RESOURCE_TYPE topCFB1
  (* Standard: 61499-2 *)
  (* Version 0.1, 2017-00-09, Hammond, HAMMONDSDESKTOP *)
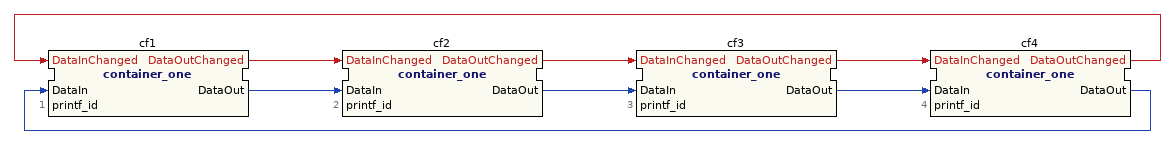
  FBS
    cf1 : container_one(printf_id := 1);
    cf2 : container_one(printf_id := 2);
    cf3 : container_one(printf_id := 3);
    cf4 : container_one(printf_id := 4);
  END_FBS
  EVENT_CONNECTIONS
    cf1.DataOutChanged TO cf2.DataInChanged;
    cf2.DataOutChanged TO cf3.DataInChanged;
    cf3.DataOutChanged TO cf4.DataInChanged;
    cf4.DataOutChanged TO cf1.DataInChanged;
  END_CONNECTIONS
  DATA_CONNECTIONS
    cf1.DataOut TO cf2.DataIn;
    cf2.DataOut TO cf3.DataIn;
    cf3.DataOut TO cf4.DataIn;
    cf4.DataOut TO cf1.DataIn;
  END_CONNECTIONS
END_RESOURCE_TYPE
